FUNCTION_BLOCK TRANS_ASE (* Composite Function Block Type *)
  (* Standard: 61499-2 *)
  (* Version 0.2, 2003-12-05, JHC, Rockwell Automation, Renamed from NEWCOMPFB. *)
  (* Version 0.1, 2002-01-08, JHC, Rockwell Automation, Added DLY FB as example. *)
  (* Version 0.0, 2000-05-27, JHC, Rockwell Automation *)
  (* Compiler header: package fb.rt.student; *)
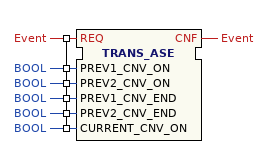
  EVENT_INPUT
    REQ WITH PREV1_CNV_ON, PREV2_CNV_ON, PREV1_CNV_END, PREV2_CNV_END, CURRENT_CNV_ON; (* Normal Execution Request *)
  END_EVENT
  EVENT_OUTPUT
    CNF; (* Execution Confirmation *)
  END_EVENT
  VAR_INPUT
    PREV1_CNV_ON : BOOL;
    PREV2_CNV_ON : BOOL;
    PREV1_CNV_END : BOOL;
    PREV2_CNV_END : BOOL;
    CURRENT_CNV_ON : BOOL;
  END_VAR
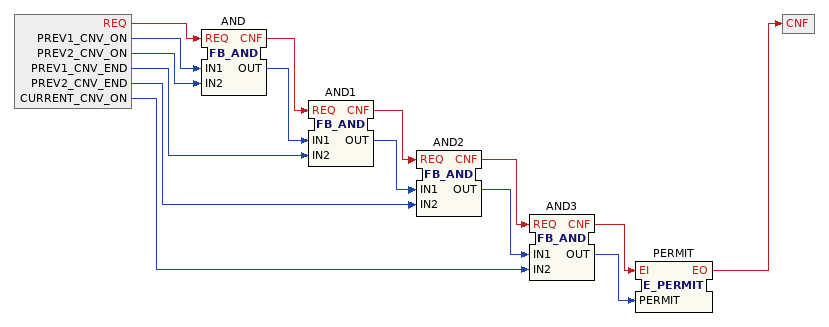
  FBS
    AND : FB_AND;
    AND1 : FB_AND;
    AND2 : FB_AND;
    AND3 : FB_AND;
    PERMIT : E_PERMIT;
  END_FBS
  EVENT_CONNECTIONS
    AND.CNF TO AND1.REQ;
    AND1.CNF TO AND2.REQ;
    AND2.CNF TO AND3.REQ;
    AND3.CNF TO PERMIT.EI;
    PERMIT.EO TO CNF;
    REQ TO AND.REQ;
  END_CONNECTIONS
  DATA_CONNECTIONS
    PREV1_CNV_ON TO AND.IN1;
    PREV2_CNV_ON TO AND.IN2;
    AND.OUT TO AND1.IN1;
    PREV1_CNV_END TO AND1.IN2;
    AND1.OUT TO AND2.IN1;
    PREV2_CNV_END TO AND2.IN2;
    AND2.OUT TO AND3.IN1;
    CURRENT_CNV_ON TO AND3.IN2;
    AND3.OUT TO PERMIT.PERMIT;
  END_CONNECTIONS
END_FUNCTION_BLOCK
